PROGRAM PB_TestRunner
VAR
    Test_LicenceCheck : TTest_LicenceCheck;
END_VAR

TcUnit.RUN();

END_PROGRAM

(* stored: Version 1.1.0.1, ProductVersion 3.1.4024.3
   POU PB_TestRunner: Id {5a6e8b50-8dd8-4eba-9459-28fa6c7e6d6e}, SpecialFunc None *)
